Staubli VAL3: RemoteAxisCtrl.dtx

bool bABSOLUTE = true
bool bBLOQ_CTRL
bool bBusy
bool bError
bool bHoming = true
bool bNewMove
bool bSTOP = true
bool bSync = true
dio Electrovalvule[2]
  [0] = {link=valve1}
  [1] = {link=valve2}
dio dBIO_salidas[4]
  [0] = {link=BasicIO-1\%Q0}
  [1] = {link=BasicIO-1\%Q1}
  [2] = {link=BasicIO-1\%Q2}
  [3] = {link=BasicIO-1\%Q3}
jointRx home = {j2=60, j3=60, j5=60}
jointRx jActualPos = {j2=60, j3=60, j5=60}
jointRx jError = {j1=0.1, j2=0.1, j3=0.1, j4=0.1, j5=0.1, j6=0.1}
jointRx jdestino = {j2=60, j3=60, j5=60}
jointRx origen
mdesc mNomSpeed = {blend=off}
mdesc mSpeed = {vel=10, blend=off}
num action
num axis_v[6]
  [5] = 1
num d_min = 0.5
num error_code
num g_data[82]
  [0] = 156
  [1] = 124
  [2] = 66
  [3] = 89
  [4] = 39
  [5] = 121
  [6] = 244
  [7] = 77
  [12] = 66
  [18] = 128
  [20] = 20
  [21] = 10
  [42] = 100
num g_message_send[82]
  [0] = 156
  [1] = 124
  [2] = 66
  [3] = 89
  [4] = 39
  [5] = 121
  [6] = 244
  [7] = 77
  [12] = 66
  [16] = 32
  [20] = 20
  [21] = 10
  [22] = 250
  [23] = 202
  [26] = 208
  [27] = 7
  [30] = 64
  [31] = 31
  [34] = 80
  [35] = 70
  [42] = 80
  [43] = 70
  [48] = 1
  [49] = 1
  [51] = 1
num id = -1
num id_actual = -2
num joint_v[6]
num mode_mov
num move_inc = 1
num nBytes
num n_status = 1
num speed = 10
num working_mode
pointRx pActualPos = {x=519.615242, y=20, z=-80, rx=-180, rz=-180, shoulder=lefty, elbow=epositive, wrist=wpositive, fatherId=world[0]}
pointRx pPunto = {fatherId=world[0]}
pointRx pdestino = {x=539.615242, y=40, z=-60, rx=-160, ry=20, rz=-160, shoulder=lefty, elbow=epositive, wrist=wpositive, fatherId=world[0]}
sio sSockPC = {link=Socket\RemoteCTRL}
tool tGripper = {fatherId=flange[0], ioLink=valve1}
